FUNCTION_BLOCK FB_GCodeTool EXTENDS FB_MzTool
VAR_INPUT
END_VAR
VAR_OUTPUT
END_VAR
VAR
	nGCodeToolNr : USINT;
END_VAR

SUPER^();	//FB_MzTool aufrufen

METHOD M_CheckGCodeStart : ERRORID
VAR_INPUT
END_VAR
//Wird derzeit von den Tool überschrieben, die Extruder sind und gelockt werden müssen.
END_METHOD

METHOD M_GetAllProps : ERRORID
VAR_INPUT
	refCmdData : REFERENCE TO  ST_CmdData;
END_VAR
SUPER^.M_GetAllProps(refCmdData);
nCurrentPropIndex := nCurrentPropIndex + 1;
refCmdData.n32Data[nCurrentPropIndex] := nGCodeToolNr;
END_METHOD

METHOD M_SetAllProps : ERRORID
VAR_INPUT
	refCmdData : REFERENCE TO  ST_CmdData;
END_VAR
M_SetAllProps := SUPER^.M_SetAllProps(refCmdData);

IF M_SetAllProps > 0 THEN
	RETURN;
END_IF

nCurrentPropIndex := nCurrentPropIndex + 1;
nSpecPropIndex := nCurrentPropIndex;
nGCodeToolNr := DINT_TO_USINT(refCmdData.n32Data[nCurrentPropIndex]);
nNoOfProps := nCurrentPropIndex + 1;

eObjectGroup := eObjectGroup OR E_ObjectGroup.OBJECTGROUP_GCodeTool;
END_METHOD

METHOD M_SetPrintParams : ST_MethResult
VAR_INPUT
	eType 		: E_PrintParamType;
	nNumerator	: USINT;
	nValue		: DINT;
END_VAR
END_METHOD

METHOD M_StartUniDispense : ERRORID
VAR_INPUT
	nParam1 : DINT;
	nParam2 : DINT;
END_VAR

VAR_OUTPUT
	bIsContinous : BOOL;
END_VAR
M_StartUniDispense := E_ErrorIdGCode.ERRORID_ToolIsNoUniDispenser;
END_METHOD

METHOD M_StopUniDispense : ERRORID
VAR_INPUT
END_VAR
END_METHOD

PROPERTY P_nGCodeToolNr : USINT
GET
P_nGCodeToolNr := nGCodeToolNr;
END_GET
END_PROPERTY

END_FUNCTION_BLOCK

(* stored: Version 1.1.0.1, ProductVersion 3.1.4024.9
   POU FB_GCodeTool: Id {c75034e7-4234-4670-b0af-42a8f7aa99d4}, SpecialFunc None
   Method M_CheckGCodeStart: Id {3f37db1e-b851-472c-b204-51f43e64851d}
   Method M_GetAllProps: Id {4539080a-72d4-4352-bdd7-c7e8557154d6}
   Method M_SetAllProps: Id {1a22e44e-fd1e-42a0-a6db-60829e335169}
   Method M_SetPrintParams: Id {0f43d903-a594-446c-864c-b193be8f1ac6}
   Method M_StartUniDispense: Id {8a621b59-82c0-4dc2-8cff-ca3062cf9646}
   Method M_StopUniDispense: Id {54aab880-5772-4aea-b02c-5f6a7f7b9cb7}
   Property P_nGCodeToolNr: Id {7a8407f9-50c9-41e9-b365-6801dac01bf6}
   Get Get: Id {6020b870-7c2b-4146-826a-d9856fc3e614} *)
